PROGRAM P_Demo_UInt64Ror
VAR
    uliHashState : T_ULARGE_INTEGER;
    dwShiftBits  : DWORD := 29;
    uliRotated   : T_ULARGE_INTEGER;
    bRotate      : BOOL;
END_VAR

// ============================================================
// Tc2_Utilities.UInt64Ror 演示程序（FUNCTION，单周期触发）
// ============================================================
// 场景：SHA-256 / SHA-512 风格哈希里的 σ₀ / σ₁ 混淆函数。
// 价值：替代 SHR+SHL+OR 三行。
// 验证步骤：
//   1. 把本 PROGRAM 加到 PlcTask 调用列表
//   2. 编译 + 登录
//   3. 在线把 b... 触发位置 TRUE 一个周期
//   4. 观察输出变量是否符合期望
// ============================================================

IF bRotate AND dwShiftBits < 64 THEN
    uliRotated := UInt64Ror(uliHashState, dwShiftBits);
    bRotate := FALSE;
END_IF;

END_PROGRAM

(* stored: Version 1.1.0.1, ProductVersion 3.1.4024.5
   POU P_Demo_UInt64Ror: Id {823c9cc1-0e95-52da-b777-a407072959ae}, SpecialFunc None *)
